TYPE (* Picture for all states *)
  (* Description: Copyright (c) 2025 HR Agrartechnik GmbH This program and the accompanying materials are made available under the terms of the Eclipse Public License 2.0 which is available at https://www.eclipse.org/legal/epl-2.0/ SPDX-License-Identifier: EPL-2.0 *)
  (* Version 1.0, 2025-06-11, Franz Höpfinger, HR Agrartechnik GmbH *)
  PACKAGE logiBUS::utils::sequence::schieber;
  IMPORT isobus::UT::Q::IDs::ID_NULL;
  SchieberStruct : STRUCT
    Unknown : UINT := ID_NULL; (* u16ObjId for Unknown State *)
    Closed : UINT := ID_NULL; (* u16ObjId for Closed State *)
    Opening : UINT := ID_NULL; (* u16ObjId for Opening State *)
    Opened : UINT := ID_NULL; (* u16ObjId for Opened State *)
    Closing : UINT := ID_NULL; (* u16ObjId for Closing State *)
  END_STRUCT;
END_TYPE
